        IF _jobNumber > inoConfig.MaxJobNumber THEN
            Messenger.Programming(_sb.Clear()
                    .Append('<#Job number (')
                    .Append(UINT_TO_STRING(_jobNumber))
                    .Append(') is greater than the maximal value of ')
                    .Append(UINT_TO_STRING(inoConfig.MaxJobNumber))
                    .Append('!#>')
                    .ToString()).Pin();

            THIS^.ThrowWhen(TRUE);
        ELSE
            _progress := _progress + 1;
        END_IF
    END_IF

    IF _progress = 2 THEN
        THIS^.inoStatus.ActionDescription :=
            _sb.Clear().Append('<#Change job by number (').Append(UINT_TO_STRING(THIS^._jobNumber)).Append(') is running.#>').ToString();

        THIS^.Messenger.OnCondition(_infoTimer.Q).Warning('<#Waiting for the signal CommandExecuting to be reseted!#>').Pin();
        THIS^.inoIoData.InspectionControl.ExecuteCommand := FALSE;
        THIS^.inoIoData.InspectionControl.ClearError := FALSE;
        THIS^.inoIoData.AcquisitionControl.SetOffline := FALSE;

        IF NOT THIS^.inoIoData.InspectionStatus.CommandExecuting THEN
            CallTimers(FALSE);
            _progress := _progress + 1;
        END_IF
    END_IF

    IF _progress = 3 THEN
        THIS^.Messenger.OnCondition(_infoTimer.Q).Warning('<#Waiting for the signal Online to be reseted!#>').Pin();
        THIS^.inoIoData.AcquisitionControl.SetOffline := TRUE;

        IF (NOT THIS^.inoIoData.AcquisitionStatus.Online) THEN
            CallTimers(FALSE);
            _progress := _progress + 1;
        END_IF
    END_IF

    IF _progress = 4 THEN
        THIS^.Messenger.OnCondition(_infoTimer.Q).Warning('<#Waiting for the signal Error to be reseted!#>').Pin();
        THIS^.inoIoData.AcquisitionControl.SetOffline := TRUE;
        THIS^.inoIoData.InspectionControl.ExecuteCommand := FALSE;
        THIS^.inoIoData.InspectionControl.ClearError := THIS^.inoIoData.InspectionStatus.Error;

        IF NOT THIS^.inoIoData.InspectionStatus.Error THEN
            CallTimers(FALSE);
            _progress := _progress + 1;
        END_IF
    END_IF

    IF _progress = 5 THEN
        THIS^.Messenger.OnCondition(_infoTimer.Q).Warning('<#Waiting for the signal CommandComplete to be set!#>').Pin();
        THIS^.inoIoData.AcquisitionControl.SetOffline := TRUE;
        THIS^.inoIoData.CommandControl.Command := _jobNumber;
        THIS^.inoIoData.InspectionControl.ExecuteCommand := TRUE;

        IF (THIS^.inoIoData.InspectionStatus.CommandComplete AND NOT THIS^.inoIoData.InspectionStatus.CommandFailed) THEN
            CallTimers(FALSE);
            _progress := _progress + 1;
        ELSIF (THIS^.inoIoData.InspectionStatus.CommandComplete AND
            THIS^.inoIoData.InspectionStatus.CommandFailed AND
            NOT THIS^.inoIoData.InspectionStatus.CommandExecuting) THEN
            _progress := 20;
        END_IF;
    END_IF

    IF _progress = 6 THEN
        THIS^.Messenger.OnCondition(_infoTimer.Q).Warning('<#Waiting for the signal CommandComplete to be reseted!#>').Pin();
        THIS^.inoIoData.AcquisitionControl.SetOffline := TRUE;
        THIS^.inoIoData.CommandControl.Command := 0;
        THIS^.inoIoData.InspectionControl.ExecuteCommand := FALSE;

        IF (NOT THIS^.inoIoData.InspectionStatus.CommandComplete) THEN
            CallTimers(FALSE);
            _progress := _progress + 1;
        END_IF;
    END_IF

    IF _progress = 7 THEN
        THIS^.Messenger.OnCondition(_infoTimer.Q).Warning('<#Waiting for the signal Online to be set!#>').Pin();
        THIS^.inoIoData.AcquisitionControl.SetOffline := FALSE;

        IF (THIS^.inoIoData.AcquisitionStatus.Online) THEN
            CallTimers(FALSE);
            _progress := _progress + 1;
        END_IF
    END_IF

    IF _progress = 8 THEN
        THIS^.inoStatus.CurrentJobNumber := UINT_TO_INT(_jobNumber);
        THIS^.inoIoData.InspectionControl.ExecuteCommand := FALSE;
        THIS^.inoIoData.AcquisitionControl.SetOffline := FALSE;
        THIS^.inoIoData.InspectionControl.ClearError := FALSE;
        THIS^.inoIoData.CommandControl.Command := 0;
        THIS^.ThrowWhen(FALSE);
        THIS^.DoneWhen(TRUE);
        _progress := 0;
    END_IF

    IF _progress = 20 THEN
        Messenger.Error(_sb.Clear()
                .Append('<#Change job by number failed. Error code:#>')
                .Append(UINT_TO_STRING(inoIoData.InspectionStatus.ErrorCode))
                .ToString()).Pin();

        THIS^.inoIoData.InspectionControl.ExecuteCommand := FALSE;
        THIS^.inoIoData.AcquisitionControl.SetOffline := FALSE;
        THIS^.inoIoData.CommandControl.Command := 0;
        THIS^.ThrowWhen(TRUE);
        THIS^.DoneWhen(FALSE);
    END_IF

    CallTimers(TRUE);
    THIS^.ThrowWhen(_errorTimer.Q);
END_IF

METHOD CallTimers
VAR_INPUT
    inValue : BOOL;
END_VAR
_infoTimer(IN := inValue, PT := THIS^.inoConfig.InfoTime);
_errorTimer(IN := inValue, PT := THIS^.inoConfig.ErrorTime);
END_METHOD

{attribute 'hide'}
METHOD PUBLIC FB_init : BOOL
VAR_INPUT
    bInitRetains : BOOL; // if TRUE, the retain variables are initialized (warm start / cold start)
    bInCopyCode : BOOL; // if TRUE, the instance afterwards gets moved into the copy code (online change)
    ParentObject : ITcoObject;
END_VAR
END_METHOD

METHOD INTERNAL InvokeWithParameters : ITcoTaskStatus
VAR_INPUT
    inJobNumber : UINT;
END_VAR
_jobNumber := inJobNumber;
InvokeWithParameters := THIS^.Invoke();
END_METHOD

(*~
    <docu>
        <summary>
            Executes when task is aborted.
        </summary>
    </docu>
~*)
METHOD PROTECTED OnAbort
THIS^.inoStatus.ActionDescription := _sb.Clear()
    .Append('<#Change job by number (')
    .Append(UINT_TO_STRING(THIS^._jobNumber))
    .Append(') aborted, while not yet finished.#>')
    .ToString();
END_METHOD

(*~
    <docu>
        <summary>
            Executes when task reaches the ```Done``` state .
        </summary>
    </docu>
~*)
METHOD PROTECTED OnDone
THIS^.inoStatus.ActionDescription :=
    _sb.Clear().Append('<#Change job by number (').Append(UINT_TO_STRING(THIS^._jobNumber)).Append(') was completed succesfully.#>').ToString();
END_METHOD

(*~
    <docu>
        <summary>
            Executes when task reaches the ```Error``` state.
            <para>
                Do not confuse with <see cref="PlcDocu.TcoCore.TcoTask.WhileError()"/>, that is called cyclically until '''Error''' state is left.
            </para>
        </summary>
    </docu>
~*)
METHOD PROTECTED OnError
THIS^.inoStatus.ActionDescription :=
    _sb.Clear().Append('<#Change job by number (').Append(UINT_TO_STRING(THIS^._jobNumber)).Append(') finished with error.#>').ToString();
END_METHOD

METHOD PROTECTED OnStart
THIS^.inoStatus.ActionDescription :=
    _sb.Clear().Append('<#Change job by number (').Append(UINT_TO_STRING(THIS^._jobNumber)).Append(') started.#>').ToString();
END_METHOD

(*~
    <docu>
        <summary>
            Restores this instance to the Ready state. Can be called explicitly or from within one of the restore mechanisms.
            <para>
                See also <see cref="PlcDocu.TcoCore.TcoTask.AutoRestorable()"/>
            </para>
        </summary>
    </docu>
~*)
METHOD Restore : ITcoRestorable
SUPER^.Restore();
_progress := 0;
CallTimers(FALSE);
Messenger.UnPin();
END_METHOD

END_FUNCTION_BLOCK

// ---- POUs/TcoInsight/v_5_x_x/Tasks/TcoInsightClearInspectionResults_v_5_x_x.TcPOU
FUNCTION_BLOCK TcoInsightClearInspectionResults_v_5_x_x EXTENDS TcoCore.TcoTask
VAR_IN_OUT
    inoIoData : TcoInsightIO_v_5_x_x;
    inoConfig : TcoInsightConfig_v_5_x_x;
    inoStatus : TcoInsightStatus_v_5_x_x;
    inoResults : TcoInsightResults_v_5_x_x;
END_VAR
VAR
    {attribute 'hide'}
    _progress : INT := 0;
    {attribute 'hide'}
    _infoTimer : TON;
    {attribute 'hide'}
    _errorTimer : TON;
    {attribute 'hide'}
    _varInfo : __SYSTEM.VAR_INFO;
    {attribute 'hide'}
    _sb : TcoCore.StringBuilder;
END_VAR

IF Execute() THEN
    IF _progress = 0 THEN
        IF NOT __ISVALIDREF(inoIoData) THEN
            _varInfo := __VARINFO(inoIoData);
            Messenger.Programming(_sb.Clear().Append('<#Invalid reference: #>').Append(_varInfo.Symbol).ToString()).Pin();
        ELSIF NOT __ISVALIDREF(inoConfig) THEN
            _varInfo := __VARINFO(inoConfig);
            Messenger.Programming(_sb.Clear().Append('<#Invalid reference: #>').Append(_varInfo.Symbol).ToString()).Pin();
        ELSIF NOT __ISVALIDREF(inoStatus) THEN
            _varInfo := __VARINFO(inoStatus);
            Messenger.Programming(_sb.Clear().Append('<#Invalid reference: #>').Append(_varInfo.Symbol).ToString()).Pin();
        ELSIF NOT __ISVALIDREF(inoResults) THEN
            _varInfo := __VARINFO(inoResults);
            Messenger.Programming(_sb.Clear().Append('<#Invalid reference: #>').Append(_varInfo.Symbol).ToString()).Pin();
        ELSE
            _progress := _progress + 1;
        END_IF
    END_IF

    IF _progress = 1 THEN
        THIS^.inoStatus.ActionDescription := '<#Clearing result data running.#>';
        CallTimers(FALSE);
        _progress := _progress + 1;
    END_IF

    IF _progress = 2 THEN
        THIS^.inoIoData.AcquisitionControl.AcquisitionTriggerEnable := FALSE;
        THIS^.inoIoData.AcquisitionControl.AcquisitionTrigger := FALSE;
        THIS^.inoIoData.InspectionControl.AcknowledgeInspectionResults := TRUE;
        THIS^.Messenger.OnCondition(_infoTimer.Q).Warning('<#Waiting for the result data cleared!#>').Pin();
        THIS^.inoResults.InspectionId := 0;
        THIS^.inoResults.ResultCode := 0;

        IF Tc2_System.MEMSET(destAddr := ADR(THIS^.inoResults.InspectionResults), fillByte := 0, n := SIZEOF(THIS^.inoResults.InspectionResults)) > 0
            THEN
            CallTimers(FALSE);
            _progress := _progress + 1;
        END_IF
    END_IF

    IF _progress = 3 THEN
        THIS^.Messenger.OnCondition(_infoTimer.Q).Warning('<#Waiting for the signal ResultsValid reseted!#>').Pin();

        IF NOT THIS^.inoIoData.InspectionStatus.ResultsValid THEN
            CallTimers(FALSE);
            _progress := _progress + 1;
        END_IF
    END_IF

    IF _progress = 4 THEN
        THIS^.inoIoData.InspectionControl.AcknowledgeInspectionResults := FALSE;
        THIS^.DoneWhen(TRUE);
        CallTimers(FALSE);
        _progress := 0;
    END_IF

    CallTimers(TRUE);
    THIS^.ThrowWhen(_errorTimer.Q);
END_IF

METHOD CallTimers
VAR_INPUT
    inValue : BOOL;
END_VAR
_infoTimer(IN := inValue, PT := THIS^.inoConfig.InfoTime);
_errorTimer(IN := inValue, PT := THIS^.inoConfig.ErrorTime);
END_METHOD

{attribute 'hide'}
METHOD PUBLIC FB_init : BOOL
VAR_INPUT
    bInitRetains : BOOL; // if TRUE, the retain variables are initialized (warm start / cold start)
    bInCopyCode : BOOL; // if TRUE, the instance afterwards gets moved into the copy code (online change)
    ParentObject : ITcoObject;
END_VAR
END_METHOD

(*~
    <docu>
        <summary>
            Executes when task is aborted.
        </summary>
    </docu>
~*)
METHOD PROTECTED OnAbort
THIS^.inoStatus.ActionDescription := '<#Clearing of the inspection results aborted, while not yet finished.#>';
END_METHOD

(*~
    <docu>
        <summary>
            Executes when task reaches the ```Done``` state .
        </summary>
    </docu>
~*)
METHOD PROTECTED OnDone
THIS^.inoStatus.ActionDescription := '<#Clearing of the inspection results was completed succesfully.#>';
END_METHOD

(*~
    <docu>
        <summary>
            Executes when task reaches the ```Error``` state.
            <para>
                Do not confuse with <see cref="PlcDocu.TcoCore.TcoTask.WhileError()"/>, that is called cyclically until '''Error''' state is left.
            </para>
        </summary>
    </docu>
~*)
METHOD PROTECTED OnError
THIS^.inoStatus.ActionDescription := '<#Clearing of the inspection results finished with error.#>';
END_METHOD

METHOD PROTECTED OnStart
THIS^.inoStatus.ActionDescription := '<#Clearing of the inspection results started.#>';
END_METHOD

(*~
    <docu>
        <summary>
            Restores this instance to the Ready state. Can be called explicitly or from within one of the restore mechanisms.
            <para>
                See also <see cref="PlcDocu.TcoCore.TcoTask.AutoRestorable()"/>
            </para>
        </summary>
    </docu>
~*)
METHOD Restore : ITcoRestorable
SUPER^.Restore();
_progress := 0;
CallTimers(FALSE);
Messenger.UnPin();
END_METHOD

END_FUNCTION_BLOCK

// ---- POUs/TcoInsight/v_5_x_x/Tasks/TcoInsightSoftEvent_v_5_x_x.TcPOU
FUNCTION_BLOCK TcoInsightSoftEvent_v_5_x_x EXTENDS TcoCore.TcoTask
VAR_IN_OUT
    inoIoData : TcoInsightIO_v_5_x_x;
    inoConfig : TcoInsightConfig_v_5_x_x;
    inoStatus : TcoInsightStatus_v_5_x_x;
END_VAR
VAR
    {attribute addProperty Name "<#Soft event number#>"}
    _softEventNumber : UINT;
END_VAR
VAR
    {attribute 'hide'}
    _progress : INT := 0;
    {attribute 'hide'}
    _infoTimer : TON;
    {attribute 'hide'}
    _errorTimer : TON;
    {attribute 'hide'}
    _varInfo : __SYSTEM.VAR_INFO;
    {attribute 'hide'}
    _sb : TcoCore.StringBuilder;
    {attribute 'hide'}
    _inspectionCompleted : BOOL;
END_VAR

IF Execute() THEN
    IF _progress = 0 THEN
        IF NOT __ISVALIDREF(inoIoData) THEN
            _varInfo := __VARINFO(inoIoData);
            Messenger.Programming(_sb.Clear().Append('<#Invalid reference: #>').Append(_varInfo.Symbol).ToString()).Pin();
        ELSIF NOT __ISVALIDREF(inoConfig) THEN
            _varInfo := __VARINFO(inoConfig);
            Messenger.Programming(_sb.Clear().Append('<#Invalid reference: #>').Append(_varInfo.Symbol).ToString()).Pin();
        ELSIF NOT __ISVALIDREF(inoStatus) THEN
            _varInfo := __VARINFO(inoStatus);
            Messenger.Programming(_sb.Clear().Append('<#Invalid reference: #>').Append(_varInfo.Symbol).ToString()).Pin();
        ELSE
            _progress := _progress + 1;
        END_IF
    END_IF

    IF _progress = 1 THEN
        CallTimers(FALSE);

        IF _softEventNumber > 7 THEN
            Messenger.Programming(_sb.Clear()
                    .Append('<#SoftEvent number: (')
                    .Append(UINT_TO_STRING(_softEventNumber))
                    .Append(') is greater than the maximal value of 7!#>')
                    .ToString()).Pin();

            THIS^.ThrowWhen(TRUE);
        ELSE
            _progress := _progress + 1;
        END_IF
    END_IF

    IF _progress = 2 THEN
        THIS^.inoStatus.ActionDescription :=
            _sb.Clear().Append('<#SoftEvent (number: ').Append(UINT_TO_STRING(THIS^._softEventNumber)).Append(') is running.#>').ToString();

        CallTimers(FALSE);
        _progress := _progress + 1;
    END_IF

    IF _progress = 3 THEN
        THIS^.Messenger.OnCondition(_infoTimer.Q)
            .Warning(_sb.Clear()
                .Append('<#Waiting for the signal TriggerSoftEvent[')
                .Append(UINT_TO_STRING(THIS^._softEventNumber))
                .Append('] to be set!#>')
                .ToString()).Pin();

        THIS^.inoIoData.SoftEventControl.TriggerSoftEvent[_softEventNumber] := TRUE;

        IF THIS^.inoIoData.SoftEventControl.TriggerSoftEventAcknowledge[_softEventNumber] THEN
            CallTimers(FALSE);
            _progress := _progress + 1;
        END_IF
    END_IF

    IF _progress = 4 THEN
        THIS^.Messenger.OnCondition(_infoTimer.Q)
            .Warning(_sb.Clear()
                .Append('<#Waiting for the signal TriggerSoftEvent[')
                .Append(UINT_TO_STRING(THIS^._softEventNumber))
                .Append('] to be reseted!#>')
                .ToString()).Pin();

        THIS^.inoIoData.SoftEventControl.TriggerSoftEvent[_softEventNumber] := FALSE;

        IF NOT THIS^.inoIoData.SoftEventControl.TriggerSoftEventAcknowledge[_softEventNumber] THEN
            CallTimers(FALSE);
            _progress := _progress + 1;
        END_IF
    END_IF

    IF _progress = 5 THEN
        THIS^.DoneWhen(TRUE);
        _progress := 0;
    END_IF

    CallTimers(TRUE);
    THIS^.ThrowWhen(_errorTimer.Q);
END_IF

METHOD CallTimers
VAR_INPUT
    inValue : BOOL;
END_VAR
_infoTimer(IN := inValue, PT := THIS^.inoConfig.InfoTime);
_errorTimer(IN := inValue, PT := THIS^.inoConfig.ErrorTime);
END_METHOD

{attribute 'hide'}
METHOD PUBLIC FB_init : BOOL
VAR_INPUT
    bInitRetains : BOOL; // if TRUE, the retain variables are initialized (warm start / cold start)
    bInCopyCode : BOOL; // if TRUE, the instance afterwards gets moved into the copy code (online change)
    ParentObject : ITcoObject;
END_VAR
END_METHOD

METHOD INTERNAL InvokeWithParameters : ITcoTaskStatus
VAR_INPUT
    inSoftEventNumber : UINT;
END_VAR
_softEventNumber := inSoftEventNumber;
InvokeWithParameters := THIS^.Invoke();
END_METHOD

(*~
    <docu>
        <summary>
            Executes when task is aborted.
        </summary>
    </docu>
~*)
METHOD PROTECTED OnAbort
THIS^.inoStatus.ActionDescription := _sb.Clear()
    .Append('<#SoftEvent (number: ')
    .Append(UINT_TO_STRING(THIS^._softEventNumber))
    .Append(') was aborted, while not yet completed.#>')
    .ToString();
END_METHOD

(*~
    <docu>
        <summary>
            Executes when task reaches the ```Done``` state .
        </summary>
    </docu>
~*)
METHOD PROTECTED OnDone
THIS^.inoStatus.ActionDescription :=
    _sb.Clear().Append('<#SoftEvent (number: ').Append(UINT_TO_STRING(THIS^._softEventNumber)).Append(') was completed successfully.#>').ToString();
END_METHOD

(*~
    <docu>
        <summary>
            Executes when task reaches the ```Error``` state.
            <para>
                Do not confuse with <see cref="PlcDocu.TcoCore.TcoTask.WhileError()"/>, that is called cyclically until '''Error''' state is left.
            </para>
        </summary>
    </docu>
~*)
METHOD PROTECTED OnError
THIS^.inoStatus.ActionDescription :=
    _sb.Clear().Append('<#SoftEvent (number: ').Append(UINT_TO_STRING(THIS^._softEventNumber)).Append(') finished with error.#>').ToString();
END_METHOD

METHOD PROTECTED OnStart
THIS^.inoStatus.ActionDescription :=
    _sb.Clear().Append('<#SoftEvent (number: ').Append(UINT_TO_STRING(THIS^._softEventNumber)).Append(') started.#>').ToString();
END_METHOD

(*~
    <docu>
        <summary>
            Restores this instance to the Ready state. Can be called explicitly or from within one of the restore mechanisms.
            <para>
                See also <see cref="PlcDocu.TcoCore.TcoTask.AutoRestorable()"/>
            </para>
        </summary>
    </docu>
~*)
METHOD Restore : ITcoRestorable
SUPER^.Restore();
_progress := 0;
CallTimers(FALSE);
Messenger.UnPin();
END_METHOD

END_FUNCTION_BLOCK

// ---- POUs/TcoInsight/v_5_x_x/TcoInsight_v_5_x_x.TcPOU
FUNCTION_BLOCK TcoInsight_v_5_x_x EXTENDS TcoIo.TcoPnIoComponent
VAR_IN_OUT
    inoIoData : TcoInsightIO_v_5_x_x;
END_VAR
VAR
    {attribute addProperty Name "<#Config#>"}
    _config : TcoInsightConfig_v_5_x_x;
    {attribute addProperty Name "<#Status#>"}
    _status : TcoInsightStatus_v_5_x_x;
END_VAR
VAR
    {attribute addProperty Name "<#UserData#>"}
    _userData : TcoInsightUser_v_5_x_x;
    {attribute addProperty Name "<#Results#>"}
    _results : TcoInsightResults_v_5_x_x;
END_VAR
VAR
    {attribute 'hide'}
    _taskEnabled : BOOL;
    {attribute addProperty Name "<#Restore#>"}
    _restoreTask : TcoCore.TcoTask(THIS^);
    {attribute addProperty Name "<#Update signal states#>"}
    _updateSignalStatesTask : TcoCore.TcoTask(THIS^);
    {attribute addProperty Name "<#Change job by number#>"}
    _changeJobByNumberTask : TcoInsightChangeJobByNumber_v_5_x_x(THIS^);
    {attribute addProperty Name "<#Change job by name#>"}
    _changeJobByNameTask : TcoInsightChangeJobByName_v_5_x_x(THIS^);
    {attribute addProperty Name "<#Clear inspection results#>"}
    _clearInspectionResultsTask : TcoInsightClearInspectionResults_v_5_x_x(THIS^);
    {attribute addProperty Name "<#Soft event#>"}
    _softEventTask : TcoInsightSoftEvent_v_5_x_x(THIS^);
    {attribute addProperty Name "<#Trigger#>"}
    _triggerTask : TcoInsightTrigger_v_5_x_x(THIS^);
END_VAR
VAR
    {attribute 'hide'}
    _varInfo : __SYSTEM.VAR_INFO;
    {attribute 'hide'}
    _sb : TcoCore.StringBuilder;
END_VAR

IF InvalidReference() THEN
    RETURN;
END_IF

SUPER^(inPnIoBoxState := THIS^.inoIoData.PnIoBoxState, inPnIoBoxDiag := THIS^.inoIoData.PnIoBoxDiag);

IF NOT SUPER^.ProfinetReady THEN
    THIS^._status.ActionDescription := '<#Not ready for operation by means of Profinet network!#>';
END_IF

IF SUPER^.ProfinetReady AND THIS^._status.ActionDescription = '<#Not ready for operation by means of Profinet network!#>' THEN
    THIS^._status.ActionDescription := '<#Ready for operation!#>';
END_IF

CheckIfOnline();
//*************RESTORE********************
_taskEnabled := TRUE;
_restoreTask.Enabled := _taskEnabled;

IF _restoreTask.Execute() THEN
    Restore();
    //	UpdateSignalStates();
END_IF

//****************************************
//*************UPDATE*********************
IF _config.UpdateStatesPermanently THEN
    UpdateSignalStates();
END_IF;

_taskEnabled := SUPER^.ProfinetReady;
_taskEnabled := _taskEnabled AND NOT _restoreTask.Busy;
_updateSignalStatesTask.Enabled := _taskEnabled;

IF _updateSignalStatesTask.Execute() THEN
    UpdateSignalStates();
END_IF
//****************************************
//*************CHANGE*JOB*BY*NUMBER*******
_taskEnabled := SUPER^.ProfinetReady;
_taskEnabled := _taskEnabled AND NOT _updateSignalStatesTask.Busy;
_changeJobByNumberTask.Enabled := _taskEnabled;
_changeJobByNumberTask(inoIoData := THIS^.inoIoData, inoConfig := THIS^._config, inoStatus := THIS^._status);
//****************************************
//*************CHANGE*JOB*BY*NAME*********
_taskEnabled := SUPER^.ProfinetReady;
_taskEnabled := _taskEnabled AND NOT _changeJobByNumberTask.Busy;
_changeJobByNameTask.Enabled := _taskEnabled;
_changeJobByNameTask(inoIoData := THIS^.inoIoData, inoConfig := THIS^._config, inoStatus := THIS^._status);
//****************************************
//*************CLEAR*DATA*****************
_taskEnabled := SUPER^.ProfinetReady;
_taskEnabled := _taskEnabled AND NOT _changeJobByNameTask.Busy;
_clearInspectionResultsTask.Enabled := _taskEnabled;

_clearInspectionResultsTask(inoIoData := THIS^.inoIoData,
    inoConfig := THIS^._config,
    inoStatus := THIS^._status,
    inoResults := THIS^._results);
//****************************************
//*************SOFT*EVENT*****************
_taskEnabled := SUPER^.ProfinetReady;
_taskEnabled := _taskEnabled AND THIS^.inoIoData.AcquisitionStatus.Online AND NOT _clearInspectionResultsTask.Busy;
_softEventTask.Enabled := _taskEnabled;
_softEventTask(inoIoData := THIS^.inoIoData, inoConfig := THIS^._config, inoStatus := THIS^._status);
//****************************************
//*************TRIGGER********************
_taskEnabled := SUPER^.ProfinetReady;
_taskEnabled := _taskEnabled AND NOT _clearInspectionResultsTask.Busy;
_triggerTask.Enabled := _taskEnabled;

_triggerTask(inoIoData := THIS^.inoIoData,
    inoConfig := THIS^._config,
    inoStatus := THIS^._status,
    inoResults := THIS^._results);
//****************************************

(*~
    <docu>
        <summary>
            Clears the inspection results.
        </summary>
    </docu>
~*)
METHOD ClearInspectionResults : TcoCore.ITcoTaskStatus
ClearInspectionResults := THIS^._clearInspectionResultsTask.Invoke();
END_METHOD

(*~
    <docu>
        <summary>
            Gets the `ClearResultDataTask` task that controls clearing of the results data.
        </summary>
    </docu>
~*)
PROPERTY ClearInspectionResultsTask : TcoCore.ITcoTaskStatus
GET
ClearInspectionResultsTask := THIS^._clearInspectionResultsTask;
END_GET
END_PROPERTY

(*~
    <docu>
        <summary>
            Gets the configuration of the sensor.
        </summary>
    </docu>
~*)
PROPERTY Config : REFERENCE TO TcoInsightConfig_v_5_x_x
GET
Config REF= _config;
END_GET
END_PROPERTY

METHOD FB_init : BOOL
VAR_INPUT
    bInitRetains : BOOL; // if TRUE, the retain variables are initialized (warm start / cold start)
    bInCopyCode : BOOL; // if TRUE, the instance afterwards gets moved into the copy code (online change)
    ParentObject : ITcoObject;
END_VAR
END_METHOD

METHOD GetResultAsByte : BYTE
VAR_INPUT
    inPosition : UINT;
END_VAR
VAR
    _size : UINT;
END_VAR
_size := SIZEOF(GetResultAsByte);

IF (inPosition + _size) > THIS^._config.ResultDataSize THEN
    Messenger.Warning('<#Index of the ResultData in the method GetResultAsByte exceeds the size hardware structure mapped!#>');
    RETURN;
END_IF

IF (inPosition + _size) > TcoVisionParams.MAX_BYTE_ARRAY THEN
    Messenger.Programming('<#Index of the ResultData in the method GetResultAsByte exceeds the defined size!#>');
    RETURN;
END_IF

GetResultAsByte := THIS^._results.InspectionResults[inPosition];
END_METHOD

METHOD GetResultAsDint : DINT
VAR_INPUT
    inPosition : UINT;
END_VAR
VAR
    _index : UINT;
    _size : UINT;
END_VAR
_size := SIZEOF(GetResultAsDint);

IF (inPosition + _size) > THIS^._config.ResultDataSize THEN
    Messenger.Warning('<#Index of the ResultData in the method GetResultAsDint exceeds the size hardware structure mapped!#>');
    RETURN;
END_IF

IF (inPosition + _size) > TcoVisionParams.MAX_BYTE_ARRAY THEN
    Messenger.Programming('<#Index of the ResultData in the method GetResultAsDint exceeds the defined size!#>');
    RETURN;
END_IF

GetResultAsDint := TcoUtilities.TcoBytesToDint(THIS^._config.DataFormat,
    THIS^._results.InspectionResults[inPosition],
    THIS^._results.InspectionResults[inPosition + 1],
    THIS^._results.InspectionResults[inPosition + 2],
    THIS^._results.InspectionResults[inPosition + 3]);
END_METHOD

METHOD GetResultAsReal : REAL
VAR_INPUT
    inPosition : UINT;
END_VAR
VAR
    _index : UINT;
    _size : UINT;
END_VAR
_size := SIZEOF(GetResultAsReal);

IF (inPosition + _size) > THIS^._config.ResultDataSize THEN
    Messenger.Warning('<#Index of the ResultData in the method GetResultAsReal exceeds the size hardware structure mapped!#>');
    RETURN;
END_IF

IF (inPosition + _size) > TcoVisionParams.MAX_BYTE_ARRAY THEN
    Messenger.Programming('<#Index of the ResultData in the method GetResultAsReal exceeds the defined size!#>');
    RETURN;
END_IF

GetResultAsReal := TcoUtilities.TcoBytesToReal(THIS^._config.DataFormat,
    THIS^._results.InspectionResults[inPosition],
    THIS^._results.InspectionResults[inPosition + 1],
    THIS^._results.InspectionResults[inPosition + 2],
    THIS^._results.InspectionResults[inPosition + 3]);
END_METHOD

METHOD GetResultAsString : STRING
VAR_INPUT
    inPosition : UINT;
    inLength : UINT;
END_VAR
VAR
    _index : UINT;
    _bufferSize : UINT;
    _resultString : STRING;
END_VAR
IF (inPosition + inLength) > THIS^._config.ResultDataSize THEN
    Messenger.Warning('<#Index of the ResultData in the method GetResultAsString exceeds the size hardware structure mapped!#>');
    RETURN;
END_IF

IF (inPosition + inLength) > TcoVisionParams.MAX_BYTE_ARRAY THEN
    Messenger.Programming('<#Index of the ResultData in the method GetResultAsString exceeds the defined size!#>');
    RETURN;
END_IF

_resultString := '';

IF (inLength > 0) THEN
    FOR _index := 0 TO inLength - 1 BY 1 DO
        IF (THIS^._results.InspectionResults[inPosition + _index] <> 0) THEN
            _resultString := CONCAT(_resultString, F_ToCHR(THIS^._results.InspectionResults[inPosition + _index]));
        ELSE
            EXIT;
        END_IF
    END_FOR;
END_IF

GetResultAsString := _resultString;
END_METHOD

(*~
    <docu>
        <summary>
            Changes the job by its name.
        </summary>
    </docu>
~*)
METHOD ChangeJobByName : TcoCore.ITcoTaskStatus
VAR_INPUT
    inJobName : STRING;
END_VAR
ChangeJobByName := THIS^._changeJobByNameTask.InvokeWithParameters(inJobName);
END_METHOD

(*~
    <docu>
        <summary>
            Gets the `ClearResultDataTask` task that controls clearing of the results data.
        </summary>
    </docu>
~*)
PROPERTY ChangeJobByNameTask : TcoCore.ITcoTaskStatus
GET
ChangeJobByNameTask := THIS^._changeJobByNameTask;
END_GET
END_PROPERTY

(*~
    <docu>
        <summary>
            Changes the job by its identification number.
        </summary>
    </docu>
~*)
METHOD ChangeJobByNumber : TcoCore.ITcoTaskStatus
VAR_INPUT
    inJobNumber : UINT;
END_VAR
ChangeJobByNumber := THIS^._changeJobByNumberTask.InvokeWithParameters(inJobNumber);
END_METHOD

(*~
    <docu>
        <summary>
            Gets the `ClearResultDataTask` task that controls clearing of the results data.
        </summary>
    </docu>
~*)
PROPERTY ChangeJobByNumberTask : TcoCore.ITcoTaskStatus
GET
ChangeJobByNumberTask := THIS^._changeJobByNumberTask;
END_GET
END_PROPERTY

METHOD INTERNAL CheckIfOnline
VAR_INST
    _onlineTimer : TON;
END_VAR
IF NOT THIS^.inoIoData.AcquisitionStatus.Online THEN
    THIS^._status.CurrentJobName := '';
    THIS^._status.CurrentJobNumber := -1;
END_IF

_onlineTimer(IN := NOT THIS^.inoIoData.AcquisitionControl.SetOffline AND NOT THIS^.inoIoData.AcquisitionStatus.Online, PT := T#3S);

Messenger.OnCondition(inoIoData.AcquisitionStatus.OfflineReason0 AND _onlineTimer.Q)
    .Info('<#Camera offline:The vision system$'s job is being modified.#>');

Messenger.OnCondition(inoIoData.AcquisitionStatus.OfflineReason0 AND _onlineTimer.Q)
    .Info('<#Camera offline:A discrete signal is holding the vision system Offline.#>');

Messenger.OnCondition(inoIoData.AcquisitionStatus.OfflineReason0 AND _onlineTimer.Q)
    .Info('<#Camera offline:A communications protocol is holding the vision system Offline.#>');
END_METHOD

METHOD INTERNAL InvalidReference : BOOL
InvalidReference := FALSE;

IF NOT __ISVALIDREF(inoIoData) THEN
    _varInfo := __VARINFO(inoIoData);
    Messenger.Programming(_sb.Clear().Append('<#Invalid reference: #>').Append(_varInfo.Symbol).ToString());
    InvalidReference := TRUE;
END_IF
END_METHOD

PROPERTY LastResultData : TcoInsightResults_v_5_x_x
GET
LastResultData := THIS^._results;
END_GET
END_PROPERTY

(*~
    <docu>
        <summary>
            Restores this instance to the Ready state. Can be called explicitly or from within one of the restore mechanisms.
        </summary>
    </docu>
~*)
METHOD Restore : ITcoRestorable
_updateSignalStatesTask.Restore();
_changeJobByNumberTask.Restore();
_changeJobByNameTask.Restore();
_clearInspectionResultsTask.Restore();
_softEventTask.Restore();
_triggerTask.Restore();
Tc2_System.MEMSET(destAddr := ADR(THIS^._results.InspectionResults), fillByte := 0, n := SIZEOF(THIS^._results.InspectionResults));
THIS^._results.InspectionId := 0;
THIS^._results.ResultCode := 0;

IF InvalidReference() THEN
    RETURN;
END_IF

Tc2_System.MEMSET(destAddr := ADR(THIS^.inoIoData), fillByte := 0, n := SIZEOF(THIS^.inoIoData));
_status.ActionDescription := '<#Restore executed!#>';
_restoreTask.Restore();
END_METHOD

(*~
    <docu>
        <summary>
            Custom service (manual, maintenance) logic.
            This method must be implemented in derived class.
        </summary>
    </docu>
~*)
METHOD PROTECTED ServiceMode
END_METHOD

METHOD SetUserDataAsByte : BOOL;
VAR_INPUT
    inValue : BYTE;
    inPosition : UINT;
END_VAR
VAR
    _bufferSize : UINT;
    _size : UINT;
END_VAR
SetUserDataAsByte := FALSE;
_size := SIZEOF(inValue);
_bufferSize := SIZEOF(THIS^._userData.UserData) / SIZEOF(THIS^._userData.UserData[0]);

IF (inPosition + _size) > THIS^._config.UserDataSize THEN
    Messenger.Info('<#Index of UserData in method SetUserDataAsByte exceeds the size hardware structure mapped#>');
    RETURN;
END_IF

IF (inPosition + _size) > _bufferSize THEN
    Messenger.Info('<#Index of UserData in method SetUserDataAsByte exceeds the defined size#>');
    RETURN;
END_IF

THIS^._userData.UserData[inPosition] := inValue;
SetUserDataAsByte := TRUE;
END_METHOD

METHOD SetUserDataAsDint : BOOL
VAR_INPUT
    inValue : DINT;
    inPosition : UINT;
END_VAR
VAR
    _index : UINT;
    _size : UINT;
    _bufferSize : UINT;
END_VAR
SetUserDataAsDint := FALSE;
_size := SIZEOF(inValue);
_bufferSize := SIZEOF(THIS^._userData.UserData) / SIZEOF(THIS^._userData.UserData[0]);

IF (inPosition + _size) > THIS^._config.UserDataSize THEN
    Messenger.Info('<#Index of UserData in method SetUserDataAsDint exceeds the size hardware structure mapped#>');
    RETURN;
END_IF

IF (inPosition + _size) > _bufferSize THEN
    Messenger.Info('<#Index of UserData in method SetUserDataAsDint exceeds the defined size#>');
    RETURN;
END_IF

TcoDintToBytes(THIS^._config.DataFormat,
    inValue,
    _userData.UserData[inPosition],
    _userData.UserData[inPosition + 1],
    _userData.UserData[inPosition + 2],
    _userData.UserData[inPosition + 3]);

SetUserDataAsDint := TRUE;
END_METHOD

METHOD SetUserDataAsReal : BOOL
VAR_INPUT
    inValue : DINT;
    inPosition : UINT;
END_VAR
VAR
    _index : UINT;
    _size : UINT;
    _bufferSize : UINT;
END_VAR
SetUserDataAsReal := FALSE;
_size := SIZEOF(inValue);
_bufferSize := SIZEOF(THIS^._userData.UserData) / SIZEOF(THIS^._userData.UserData[0]);

IF (inPosition + _size) > THIS^._config.UserDataSize THEN
    Messenger.Info('<#Index of UserData in method SetUserDataAsReal exceeds the size hardware structure mapped#>');
    RETURN;
END_IF

IF (inPosition + _size) > _bufferSize THEN
    Messenger.Info('<#Index of UserData in method SetUserDataAsReal exceeds the defined size#>');
    RETURN;
END_IF

TcoRealToBytes(THIS^._config.DataFormat,
    inValue,
    _userData.UserData[inPosition],
    _userData.UserData[inPosition + 1],
    _userData.UserData[inPosition + 2],
    _userData.UserData[inPosition + 3]);

SetUserDataAsReal := TRUE;
END_METHOD

METHOD SetUserDataAsString : BOOL
VAR_INPUT
    inValue : STRING;
    inPosition : UINT;
END_VAR
VAR
    _index : UINT;
    _size : UINT;
    _bufferSize : UINT;
END_VAR
SetUserDataAsString := FALSE;
_size := LEN(inValue);
_bufferSize := SIZEOF(THIS^._userData.UserData) / SIZEOF(THIS^._userData.UserData[0]);

IF (inPosition + _size) > THIS^._config.UserDataSize THEN
    Messenger.Info('<#Index of UserData in method SetUserDataAsString exceeds the size hardware structure mapped#>');
    RETURN;
END_IF

IF (inPosition + _size) > _bufferSize THEN
    Messenger.Info('<#Index of UserData in method SetUserDataAsString exceeds the defined size#>');
    RETURN;
END_IF

FOR _index := 1 TO _size BY 1 DO
    _userData.UserData[inPosition + _index - 1] := F_ToASC(MID(inValue, 1, _index));
END_FOR;

FOR _index := inPosition + _size TO _bufferSize BY 1 DO
    _userData.UserData[_index] := 0;
END_FOR;

SetUserDataAsString := TRUE;
END_METHOD

(*~
    <docu>
        <summary>
            Executes the soft event.
        </summary>
    </docu>
~*)
METHOD SoftEvent : TcoCore.ITcoTaskStatus
VAR_INPUT
    inSoftEventNumber : UINT;
END_VAR
SoftEvent := THIS^._softEventTask.InvokeWithParameters(inSoftEventNumber);
END_METHOD

(*~
    <docu>
        <summary>
            Gets the `ClearResultDataTask` task that controls clearing of the results data.
        </summary>
    </docu>
~*)
PROPERTY SoftEventTask : TcoCore.ITcoTaskStatus
GET
SoftEventTask := THIS^._softEventTask;
END_GET
END_PROPERTY

(*~
    <docu>
        <summary>
            Gets the status of the sensor.
        </summary>
    </docu>
~*)
PROPERTY Status : REFERENCE TO TcoInsightStatus_v_5_x_x
GET
Status REF= _status;
END_GET
END_PROPERTY

(*~
    <docu>
        <summary>
            Triggers the reading sequence and waits for results.
        </summary>
    </docu>
~*)
METHOD Trigger : TcoCore.ITcoTaskStatus
Trigger := THIS^._triggerTask.Invoke();
END_METHOD

(*~
    <docu>
        <summary>
            Gets the `ClearResultDataTask` task that controls clearing of the results data.
        </summary>
    </docu>
~*)
PROPERTY TriggerTask : TcoCore.ITcoTaskStatus
GET
TriggerTask := THIS^._triggerTask;
END_GET
END_PROPERTY

METHOD INTERNAL UpdateSignalStates
_status.SignalStatus.AcquisitionTriggerEnable := inoIoData.AcquisitionControl.AcquisitionTriggerEnable;
_status.SignalStatus.AcquisitionTrigger := inoIoData.AcquisitionControl.AcquisitionTrigger;
_status.SignalStatus.ClearExposureComplete := inoIoData.AcquisitionControl.ClearExposureComplete;
_status.SignalStatus.SetOffline := inoIoData.AcquisitionControl.SetOffline;
_status.SignalStatus.EnableResultsBuffering := inoIoData.InspectionControl.EnableResultsBuffering;
_status.SignalStatus.AcknowledgeInspectionResults := inoIoData.InspectionControl.AcknowledgeInspectionResults;
_status.SignalStatus.ExtendedUserDataSet := inoIoData.InspectionControl.ExtendedUserDataSet;
_status.SignalStatus.ExecuteCommand := inoIoData.InspectionControl.ExecuteCommand;
_status.SignalStatus.ClearError := inoIoData.InspectionControl.ClearError;
_status.SignalStatus.Command := inoIoData.CommandControl.Command;
_status.SignalStatus.TriggerSoftEvent.0 := inoIoData.SoftEventControl.TriggerSoftEvent[0];
_status.SignalStatus.TriggerSoftEvent.1 := inoIoData.SoftEventControl.TriggerSoftEvent[1];
_status.SignalStatus.TriggerSoftEvent.2 := inoIoData.SoftEventControl.TriggerSoftEvent[2];
_status.SignalStatus.TriggerSoftEvent.3 := inoIoData.SoftEventControl.TriggerSoftEvent[3];
_status.SignalStatus.TriggerSoftEvent.4 := inoIoData.SoftEventControl.TriggerSoftEvent[4];
_status.SignalStatus.TriggerSoftEvent.5 := inoIoData.SoftEventControl.TriggerSoftEvent[5];
_status.SignalStatus.TriggerSoftEvent.6 := inoIoData.SoftEventControl.TriggerSoftEvent[6];
_status.SignalStatus.TriggerSoftEvent.7 := inoIoData.SoftEventControl.TriggerSoftEvent[7];
_status.SignalStatus.AcquisitionTriggerReady := inoIoData.AcquisitionStatus.AcquisitionTriggerReady;
_status.SignalStatus.AcquisitionTriggerAcknowledge := inoIoData.AcquisitionStatus.AcquisitionTriggerAcknowledge;
_status.SignalStatus.ExposureComplete := inoIoData.AcquisitionStatus.ExposureComplete;
_status.SignalStatus.MissedAcquisition := inoIoData.AcquisitionStatus.MissedAcquisition;
_status.SignalStatus.OfflineReason0 := inoIoData.AcquisitionStatus.OfflineReason0;
_status.SignalStatus.OfflineReason1 := inoIoData.AcquisitionStatus.OfflineReason1;
_status.SignalStatus.OfflineReason2 := inoIoData.AcquisitionStatus.OfflineReason2;
_status.SignalStatus.Online := inoIoData.AcquisitionStatus.Online;
_status.SignalStatus.AcquisitionID := inoIoData.AcquisitionStatus.AcquisitionID;
_status.SignalStatus.SystemBusy := inoIoData.InspectionStatus.SystemBusy;
_status.SignalStatus.InspectionCompleted := inoIoData.InspectionStatus.InspectionCompleted;
_status.SignalStatus.ResultsBufferOverrun := inoIoData.InspectionStatus.ResultsBufferOverrun;
_status.SignalStatus.ResultsValid := inoIoData.InspectionStatus.ResultsValid;
_status.SignalStatus.CommandExecuting := inoIoData.InspectionStatus.CommandExecuting;
_status.SignalStatus.CommandComplete := inoIoData.InspectionStatus.CommandComplete;
_status.SignalStatus.CommandFailed := inoIoData.InspectionStatus.CommandFailed;
_status.SignalStatus.ExtendedUserDataSetAcknowledge := inoIoData.InspectionStatus.ExtendedUserDataSetAcknowledge;
_status.SignalStatus.OverallJobPassFail := inoIoData.InspectionStatus.OverallJobPassFail;
_status.SignalStatus.TestRunReady := inoIoData.InspectionStatus.TestRunReady;
_status.SignalStatus.Error := inoIoData.InspectionStatus.Error;
_status.SignalStatus.ErrorCode := inoIoData.InspectionStatus.ErrorCode;
_status.SignalStatus.CurrentJobID := inoIoData.CommandControl.CurrentJobID;
_status.SignalStatus.TriggerSoftEventAcknowledge.0 := inoIoData.SoftEventControl.TriggerSoftEventAcknowledge[0];
_status.SignalStatus.TriggerSoftEventAcknowledge.1 := inoIoData.SoftEventControl.TriggerSoftEventAcknowledge[1];
_status.SignalStatus.TriggerSoftEventAcknowledge.2 := inoIoData.SoftEventControl.TriggerSoftEventAcknowledge[2];
_status.SignalStatus.TriggerSoftEventAcknowledge.3 := inoIoData.SoftEventControl.TriggerSoftEventAcknowledge[3];
_status.SignalStatus.TriggerSoftEventAcknowledge.4 := inoIoData.SoftEventControl.TriggerSoftEventAcknowledge[4];
_status.SignalStatus.TriggerSoftEventAcknowledge.5 := inoIoData.SoftEventControl.TriggerSoftEventAcknowledge[5];
_status.SignalStatus.TriggerSoftEventAcknowledge.6 := inoIoData.SoftEventControl.TriggerSoftEventAcknowledge[6];
_status.SignalStatus.TriggerSoftEventAcknowledge.7 := inoIoData.SoftEventControl.TriggerSoftEventAcknowledge[7];
_status.SignalStatus.InspectionID := inoIoData.ResultsData.InspectionID;
_status.SignalStatus.ResultCode := inoIoData.ResultsData.ResultCode;
_updateSignalStatesTask.DoneWhen(TRUE);
END_METHOD

PROPERTY UserData : TcoInsightUser_v_5_x_x
GET
UserData := _userData;
END_GET
END_PROPERTY

END_FUNCTION_BLOCK
